(* Logix 5000 project; controller PLCbox vendor 1 type 14 code 149 rev 30.11; software revision 30.01; part 3 of 3 *)
(* tags used below, declared in another part *)
   System_Timer : TIMER[100];
   tagToPi : DINT;

PROGRAM TestProgram   (* main routine Main *)
VAR
   ALARM : BOOL[256];
   ALARM2 : BOOL[256];
   ALARM_DESC : String20;
   ALARM_DESCR : String20[256] := ([0] := 'Fault 0', [1] := 'Fault 1', [2] := 'Fault 2');
   EmptyString : String20;
   FaultDesc : String20 := 'Fault 1';
   FaultDesc2 : String20 := 'Fault 1';
   HMI_BOOL : BOOL[32];
   Index : DINT := 256;
   PLC_BOOL : BOOL[32];
   System_Cond : BOOL[256] := ([0] := 1);
        [0]   // Start MOTOR 1
        [1]   // MOTOR 1 At Target Speed
        [2]   // Start MOTOR 2
        [3]   // Motor 2 at Target Speed
        [4]   // Heat Boiler
        [5]   // Boiler at Temp
        [6]   // System Running
        [7]   // System FAULTED
        [8]   // System RESET
   System_INT : INT[10] := ([0] := 456, [1] := 456, [2] := 1);
   System_REAL : REAL[10] := ([0] := 54.0, [1] := 54.0, [2] := 54.0);
   System_STR : STRING[10];
   System_STRING : String20[10];
   SystemFaulted : BOOL := 1;
   SystemFaulted2 : BOOL := 1;
   SystemStart : BOOL;
   SytemReset : BOOL;
   SytemReset2 : BOOL;
END_VAR

ROUTINE _02_MOV_Instruction   (* ladder *)
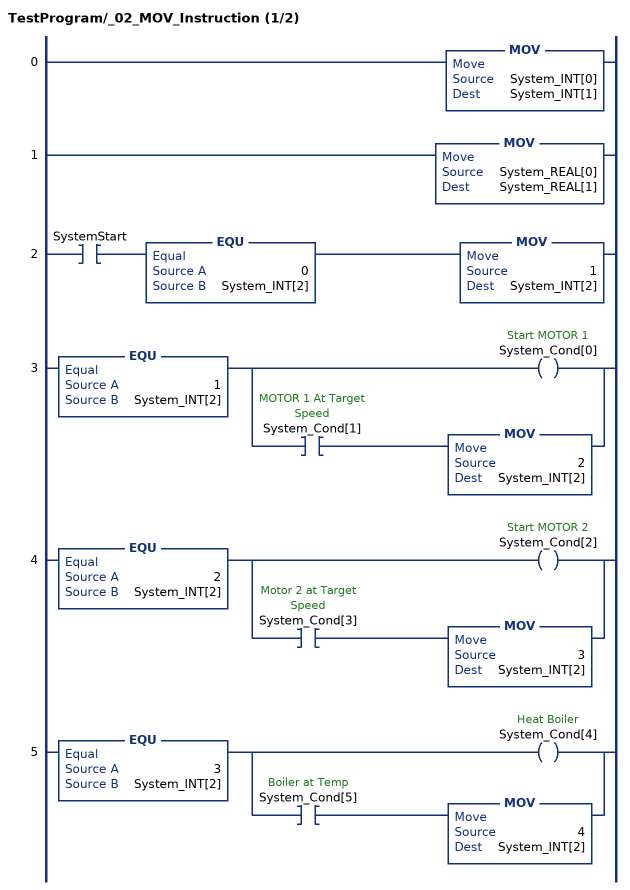
   0: MOV(System_INT[0],System_INT[1]);
   1: MOV(System_REAL[0],System_REAL[1]);
   2: XIC(SystemStart)EQU(0,System_INT[2])MOV(1,System_INT[2]);
   3: EQU(1,System_INT[2])[OTE(System_Cond[0]) ,XIC(System_Cond[1]) MOV(2,System_INT[2]) ];
   4: EQU(2,System_INT[2])[OTE(System_Cond[2]) ,XIC(System_Cond[3]) MOV(3,System_INT[2]) ];
   5: EQU(3,System_INT[2])[OTE(System_Cond[4]) ,XIC(System_Cond[5]) MOV(4,System_INT[2]) ];
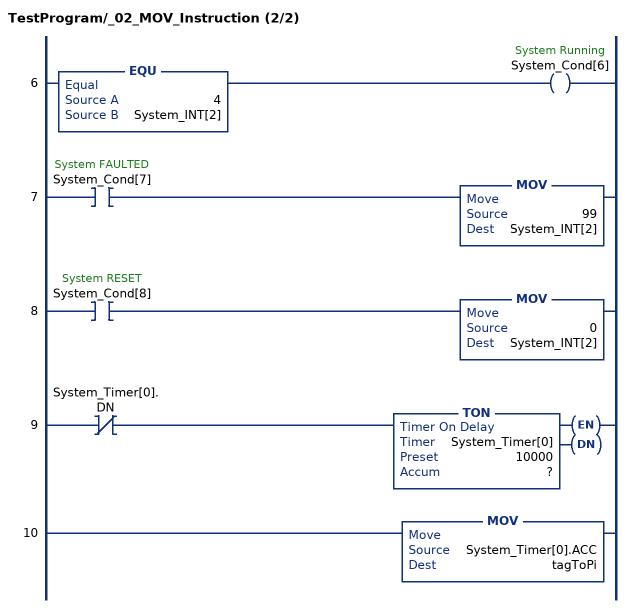
   6: EQU(4,System_INT[2])OTE(System_Cond[6]);
   7: XIC(System_Cond[7])MOV(99,System_INT[2]);
   8: XIC(System_Cond[8])MOV(0,System_INT[2]);
   9: XIO(System_Timer[0].DN)TON(System_Timer[0],?,?);
   10: MOV(System_Timer[0].ACC,tagToPi);
END_ROUTINE

ROUTINE _03_HMI   (* ladder *)
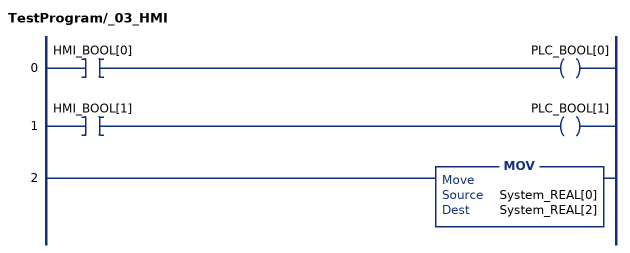
   0: XIC(HMI_BOOL[0])OTE(PLC_BOOL[0]);
   1: XIC(HMI_BOOL[1])OTE(PLC_BOOL[1]);
   2: MOV(System_REAL[0],System_REAL[2]);
END_ROUTINE

ROUTINE Main   (* ladder *)
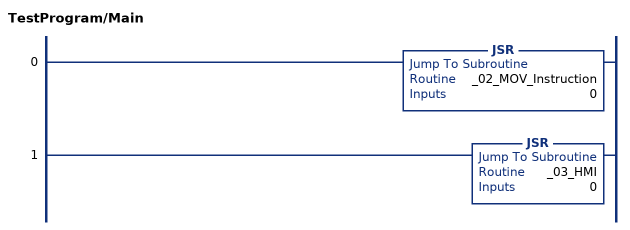
   0: JSR(_02_MOV_Instruction,0);
   1: JSR(_03_HMI,0);
END_ROUTINE
END_PROGRAM
